ABB RobotStudio station: Yumi_PCSDK_test.rsstn

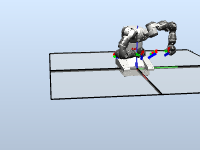
Station Yumi_PCSDK_test (saved by RobotStudio format 5)
Controller IRB_14000_0.5kg_0.5m
  mechanical unit ROB_R: IRB14000_0.5_0.5_R, 6 joints, base frame (0, 1.73, 0) mm
  mechanical unit ROB_R_7: IRB14000_0.5_0.5_R, 1 joints, base frame (0, 1.73, 0) mm
  mechanical unit ROB_L: IRB14000_0.5_0.5_L, 6 joints, base frame (0, 1.73, 0) mm
  mechanical unit ROB_L_7: IRB14000_0.5_0.5_L, 1 joints, base frame (0, 1.73, 0) mm
Layout (positions relative to the parent item):
  - IRB14000_0.5_0.5_R [mechanism, from Robots\IRB14000_0.5_0.5_R.rslib] at (0, 1.73, 0) mm; joint values [1.8779, -1.5705, -2.6481, 0.758, 2.1727, 2.3996, -1.3865] (rad or m)
  - IRB14000_0.5_0.5_L [mechanism, from Robots\IRB14000_0.5_0.5_L.rslib] at (0, 1.73, 0) mm; joint values [-0.4426, -1.633, 1.7058, 0.4713, 0.2052, 0.9717, -0.7063] (rad or m)
Targets, tools, work objects and paths stored in the station, written as RAPID:
! task T_ROB_R
MODULE Module1
  CONST robtarget Target_10:=[[109.930133311,-288.730230127,184.680148405],[0.471815059,-0.579336906,-0.624806977,-0.226661733],[0,0,0,11],[162.18999224,9E9,9E9,9E9,9E9,9E9]];
ENDMODULE

! task T_ROB_L
MODULE Module1
  CONST robtarget Target_10:=[[152.477680953,185.807759776,207.487429559],[0.367323056,0.741513173,-0.346174045,0.442035652],[-1,0,-1,11],[152.879019179,9E9,9E9,9E9,9E9,9E9]];
  CONST robtarget Target_20:=[[123.609993102,156.940165007,178.619991994],[0.367323217,0.741513338,-0.346173505,0.442035663],[-1,0,-1,11],[152.878973879,9E9,9E9,9E9,9E9,9E9]];
  PROC Path_10()
    MoveL Target_10,v1000,z100,tool0\WObj:=wobj0;
  ENDPROC
ENDMODULE

